(* IEC 61131-3 sources: volt/packages/volt-lsp-iec/test-corpus/pro2193/Device/Plc Logic/Application/99 Library/Function Blocks/JSON builders, 6 files *)

(* ---- BoxFillingJsonFB.pou ---- *)
FUNCTION_BLOCK BoxFillingJsonFB
EXTENDS ToJsonBaseFB
VAR_IN_OUT
	stacks					: ARRAY[1..GVL_Constants_BFU.MaxNumberOfStacksInBox] OF Fanuc_StackPosition;
	boxSettings				: Fanuc_BoxSettings;
	teachPosition			: Fanuc_PositionXYZWPR_Type;
	JSON					: STRING(14000);
END_VAR

%LANGUAGE ST
SUPER^();

IF busy THEN
	IF CreateFinalJson() THEN
		busy		:= FALSE;
		done		:= TRUE;
	END_IF
END_IF

END_FUNCTION_BLOCK

METHOD PRIVATE CreateBoxSettingsJson
VAR_INPUT
	pJson				: POINTER TO STRING(1);
	jsonSize			: UDINT;
END_VAR
VAR_INST
	asProperties		: ARRAY[0..10, 0..1] OF STRING(10);
END_VAR

%LANGUAGE ST
// Fill data
asProperties[0, 0]			:= 'bx';	asProperties[0, 1]			:= TO_STRING(boxSettings.BoxSize.rPosX);
asProperties[1, 0]			:= 'by';	asProperties[1, 1]			:= TO_STRING(boxSettings.BoxSize.rPosY);
asProperties[2, 0]			:= 'bz';	asProperties[2, 1]			:= TO_STRING(boxSettings.BoxSize.rPosZ);
asProperties[3, 0]			:= 'sx';	asProperties[3, 1]			:= TO_STRING(boxSettings.StackSize.rPosX);
asProperties[4, 0]			:= 'sy';	asProperties[4, 1]			:= TO_STRING(boxSettings.StackSize.rPosY);
asProperties[5, 0]			:= 'sz';	asProperties[5, 1]			:= TO_STRING(boxSettings.StackSize.rPosZ);
asProperties[6, 0]			:= 'or';	asProperties[6, 1]			:= TO_STRING(boxSettings.StackOrientation);
asProperties[7, 0]			:= 'sh';	asProperties[7, 1]			:= TO_STRING(boxSettings.StackShape);
asProperties[8, 0]			:= 'tx';	asProperties[8, 1]			:= TO_STRING(teachPosition.rPosX);
asProperties[9, 0]			:= 'ty';	asProperties[9, 1]			:= TO_STRING(teachPosition.rPosY);
asProperties[10, 0]			:= 'tz';	asProperties[10, 1]			:= TO_STRING(teachPosition.rPosZ);

CreateJson(
	psProperties				:= ADR(asProperties),
	udiPropertiesArraySize		:= SIZEOF(asProperties),
	udiPropertiesStringLength	:= SIZEOF(asProperties[0,0]),
	psJSON						:= pJson,
	udiJSONStringLength			:= jsonSize);

END_METHOD

METHOD PRIVATE CreateFinalJson : BOOL
VAR_INST
	asProperties		: ARRAY[0..GVL_Constants_BFU.MaxNumberOfStacksInBox, 0..1] OF STRING(280);
	localJSON			: STRING(14000);
END_VAR

%LANGUAGE ST
sw.Reset();

CASE chunk OF
	0:
		// Create box settings json
		sw.Start();
		asProperties[chunk, 0]	:= 'box';
		CreateBoxSettingsJson(ADR(asProperties[chunk, 1]), SIZEOF(asProperties[chunk, 1]));
		Increment.AnyInt(chunk);
		sw.End();

	1..GVL_Constants_BFU.MaxNumberOfStacksInBox:
		sw.Start();
		asProperties[chunk, 0]	:= CONCAT('S', TO_STRING(chunk));
		CreateStackJson(chunk, ADR(asProperties[chunk, 1]), SIZEOF(asProperties[chunk, 1]));
		Increment.AnyInt(chunk);
		sw.End();

	31:
		Increment.AnyInt(chunk);
	32:
		Increment.AnyInt(chunk);
	33:
		sw.Start();
		CreateJson(
			psProperties				:= ADR(asProperties),
			udiPropertiesArraySize		:= SIZEOF(asProperties),
			udiPropertiesStringLength	:= SIZEOF(asProperties[0,0]),
			psJSON						:= ADR(localJSON),
			udiJSONStringLength			:= SIZEOF(localJSON));
		sw.End();
		Increment.AnyInt(chunk);
	34:
		sw.Start();
		JSON := localJSON;
		sw.End();
		CreateFinalJson					:= TRUE;
END_CASE

END_METHOD

METHOD PRIVATE CreateStackJson
VAR_INPUT
	stack				: UINT;
	pJson				: POINTER TO STRING(1);
	jsonSize			: UDINT;
END_VAR
VAR_INST
	asProperties		: ARRAY[0..13, 0..1] OF STRING(10);
END_VAR

%LANGUAGE ST
// Fill data
asProperties[0, 0]			:= 's';		asProperties[0, 1]			:= TO_STRING(stacks[stack].StackNumber);
asProperties[1, 0]			:= 'x';		asProperties[1, 1]			:= TO_STRING(stacks[stack].PlacePosition.rPosX);
asProperties[2, 0]			:= 'y';		asProperties[2, 1]			:= TO_STRING(stacks[stack].PlacePosition.rPosY);
asProperties[3, 0]			:= 'z';		asProperties[3, 1]			:= TO_STRING(stacks[stack].PlacePosition.rPosZ);
asProperties[4, 0]			:= 'w';		asProperties[4, 1]			:= TO_STRING(stacks[stack].PlacePosition.rPosW);
asProperties[5, 0]			:= 'p';		asProperties[5, 1]			:= TO_STRING(stacks[stack].PlacePosition.rPosP);
asProperties[6, 0]			:= 'r';		asProperties[6, 1]			:= TO_STRING(stacks[stack].PlacePosition.rPosR);
asProperties[7, 0]			:= 'ox';	asProperties[7, 1]			:= TO_STRING(stacks[stack].Offset.rPosX);
asProperties[8, 0]			:= 'oy';	asProperties[8, 1]			:= TO_STRING(stacks[stack].Offset.rPosY);
asProperties[9, 0]			:= 'oz';	asProperties[9, 1]			:= TO_STRING(stacks[stack].Offset.rPosZ);
asProperties[10, 0]			:= 'tx';	asProperties[10, 1]			:= TO_STRING(stacks[stack].ToolOffset.rPosX);
asProperties[11, 0]			:= 'ty';	asProperties[11, 1]			:= TO_STRING(stacks[stack].ToolOffset.rPosY);
asProperties[12, 0]			:= 'tz';	asProperties[12, 1]			:= TO_STRING(stacks[stack].ToolOffset.rPosZ);
asProperties[13, 0]			:= 'c';		asProperties[13, 1]			:= TO_STRING(stacks[stack].Config);

CreateJson(
	psProperties				:= ADR(asProperties),
	udiPropertiesArraySize		:= SIZEOF(asProperties),
	udiPropertiesStringLength	:= SIZEOF(asProperties[0,0]),
	psJSON						:= pJson,
	udiJSONStringLength			:= jsonSize);

END_METHOD

(* ---- CassetteToJsonFB.pou ---- *)
FUNCTION_BLOCK CassetteToJsonFB
EXTENDS ToJsonBaseFB
VAR_INPUT
	CurrentDrawer			: enumDrawer;
END_VAR
VAR_IN_OUT
	CassetteDefinition		: ARRAY[1..GVL_Constants_Magazine.MaxCassettes] OF CassetteDefinition;
	TargetCassettePosition	: ARRAY[enumDrawer.Upper..enumDrawer.Lower, 1..GVL_Constants_Magazine.MaxCassettes] OF CassettePosition;
	DataCassettePosition	: ARRAY[enumDrawer.Upper..enumDrawer.Lower, 1..GVL_Constants_Magazine.MaxCassettes] OF CassettePosition;
	ActualCassettePosition	: ARRAY[enumDrawer.Upper..enumDrawer.Lower, 1..GVL_Constants_Magazine.MaxCassettes] OF CassettePosition;
	JSON					: STRING(25000);
END_VAR

%LANGUAGE ST
SUPER^();

IF busy THEN
	sw.Start();
	IF CreateFinalJson() THEN
		busy		:= FALSE;
		done		:= TRUE;
	END_IF
	sw.End();
END_IF

END_FUNCTION_BLOCK

METHOD PRIVATE CreateCassetteJson
VAR_INPUT
	cassette			: UINT;
	pJson				: POINTER TO STRING(1);
	jsonSize			: UDINT;
END_VAR
VAR_INST
	asProperties		: ARRAY[0..8, 0..1] OF STRING(50);
END_VAR

%LANGUAGE ST
// Fill data
asProperties[0, 0]		:= 'Id';	asProperties[0, 1]		:= TO_STRING(CassetteDefinition[cassette].CassetteId);
asProperties[1, 0]		:= 'Cid';	asProperties[1, 1]		:= TO_STRING(CassetteDefinition[cassette].CavityId);
asProperties[2, 0]		:= 'Lid';	asProperties[2, 1]		:= TO_STRING(CassetteDefinition[cassette].LabelId);
asProperties[3, 0]		:= 'Ltp';	asProperties[3, 1]		:= TO_STRING(CassetteDefinition[cassette].LabelType);
asProperties[4, 0]		:= 'Lor';	asProperties[4, 1]		:= TO_STRING(CassetteDefinition[cassette].LabelOrientation);
asProperties[5, 0]		:= 'Cor';	asProperties[5, 1]		:= TO_STRING(CassetteDefinition[cassette].CassetteOrientation);
asProperties[6, 0]		:= 'Act';	CreatePositionJson(position := ActualCassettePosition[	CurrentDrawer, cassette], ADR(asProperties[6, 1]), SIZEOF(asProperties[6, 1]));
asProperties[7, 0]		:= 'Tgt';	CreatePositionJson(position := TargetCassettePosition[	CurrentDrawer, cassette], ADR(asProperties[7, 1]), SIZEOF(asProperties[7, 1]));
asProperties[8, 0]		:= 'Dat';	CreatePositionJson(position := DataCassettePosition[	CurrentDrawer, cassette], ADR(asProperties[8, 1]), SIZEOF(asProperties[8, 1]));

CreateJson(
	psProperties				:= ADR(asProperties),
	udiPropertiesArraySize		:= SIZEOF(asProperties),
	udiPropertiesStringLength	:= SIZEOF(asProperties[0,0]),
	psJSON						:= pJson,
	udiJSONStringLength			:= jsonSize);

END_METHOD

METHOD PRIVATE CreateFinalJson : BOOL
VAR_INST
	asProperties		: ARRAY[1..GVL_Constants_Magazine.MaxCassettes, 0..1] OF STRING(300);
END_VAR

%LANGUAGE ST
CASE chunk OF
	0:
		Increment.AnyInt(chunk);

	1..GVL_Constants_Magazine.MaxCassettes:
		asProperties[chunk, 0]		:= CONCAT('C', TO_STRING(chunk));
		CreateCassetteJson(chunk, ADR(asProperties[chunk, 1]), SIZEOF(asProperties[chunk, 1]));
		Increment.AnyInt(chunk);

	ELSE
		CreateJson(
			psProperties				:= ADR(asProperties),
			udiPropertiesArraySize		:= SIZEOF(asProperties),
			udiPropertiesStringLength	:= SIZEOF(asProperties[1,0]),
			psJSON						:= ADR(JSON),
			udiJSONStringLength			:= SIZEOF(JSON));

		CreateFinalJson					:= TRUE;
END_CASE

END_METHOD

METHOD PRIVATE CreatePositionJson
VAR_INPUT
	position			: REFERENCE TO CassettePosition;
	pJson				: POINTER TO STRING(1);
	jsonSize			: UDINT;
END_VAR
VAR_INST
	asProperties		: ARRAY[0..2, 0..1] OF STRING(5);
END_VAR

%LANGUAGE ST
//Fill data
asProperties[0,0]		:= 'X1';	asProperties[0,1]		:= TO_STRING(position.X1);
asProperties[1,0]		:= 'X2';	asProperties[1,1]		:= TO_STRING(position.X2);
asProperties[2,0]		:= 'Y';		asProperties[2,1]		:= TO_STRING(position.Y);

CreateJson(
	psProperties				:= ADR(asProperties),
	udiPropertiesArraySize		:= SIZEOF(asProperties),
	udiPropertiesStringLength	:= SIZEOF(asProperties[0,0]),
	psJSON						:= pJson,
	udiJSONStringLength			:= jsonSize);

END_METHOD

(* ---- CavityAliasesToJsonFB.pou ---- *)
FUNCTION_BLOCK CavityAliasesToJsonFB
EXTENDS ToJsonBaseFB
VAR_IN_OUT
	aliases					: ARRAY[GVL_Constants.CavityStartIndex..GVL_Constants.CavityEndIndex] OF STRING(20);
	JSON					: STRING(2000);
END_VAR

%LANGUAGE ST
SUPER^();

IF busy THEN
	sw.Start();
	IF CreateCavityAliasJson() THEN
		busy		:= FALSE;
		done		:= TRUE;
	END_IF
	sw.End();
END_IF

END_FUNCTION_BLOCK

METHOD PRIVATE CreateCavityAliasJson  : BOOL
VAR_INST
	asProperties		: ARRAY[GVL_Constants.CavityStartIndex..GVL_Constants.CavityEndIndex, 0..1] OF STRING(20);
END_VAR

%LANGUAGE ST
// Fill data
FOR chunk := GVL_Constants.CavityStartIndex TO GVL_Constants.CavityEndIndex DO
	asProperties[chunk, 0]			:= TO_STRING(chunk);
	asProperties[chunk, 1]			:= aliases[chunk];
END_FOR

CreateJson(
	psProperties				:= ADR(asProperties),
	udiPropertiesArraySize		:= SIZEOF(asProperties),
	udiPropertiesStringLength	:= SIZEOF(asProperties[GVL_Constants.CavityStartIndex, 0]),
	psJSON						:= ADR(JSON),
	udiJSONStringLength			:= SIZEOF(JSON));

CreateCavityAliasJson			:= TRUE;

END_METHOD

(* ---- RejectReasonAliasesToJsonFB.pou ---- *)
FUNCTION_BLOCK RejectReasonAliasesToJsonFB
EXTENDS ToJsonBaseFB
VAR_IN_OUT
	aliases					: ARRAY[1..GVL_Constants.MaxRejectReasonsTotal] OF STRING(40);
	JSON					: STRING(2000);
END_VAR

%LANGUAGE ST
SUPER^();

IF busy THEN
	sw.Start();
	IF CreateRejectReasonAliasJson() THEN
		busy		:= FALSE;
		done		:= TRUE;
	END_IF
	sw.End();
END_IF

END_FUNCTION_BLOCK

METHOD PRIVATE CreateRejectReasonAliasJson : BOOL
VAR_INST
	asProperties		: ARRAY[1..GVL_Constants.MaxRejectReasonsTotal, 0..1] OF STRING(20);
END_VAR

%LANGUAGE ST
// Fill data
FOR chunk := 1 TO GVL_Constants.MaxRejectReasonsTotal DO
	asProperties[chunk, 0]			:= TO_STRING(chunk);
	asProperties[chunk, 1]			:= aliases[chunk];
END_FOR

CreateJson(
	psProperties				:= ADR(asProperties),
	udiPropertiesArraySize		:= SIZEOF(asProperties),
	udiPropertiesStringLength	:= SIZEOF(asProperties[1, 0]),
	psJSON						:= ADR(JSON),
	udiJSONStringLength			:= SIZEOF(JSON));

CreateRejectReasonAliasJson		:= TRUE;

END_METHOD

(* ---- StatsToJsonFB.pou ---- *)
FUNCTION_BLOCK StatsToJsonFB
EXTENDS ToJsonBaseFB
VAR_IN_OUT
	stats					: ProductionStatsType;
	JSON					: STRING(25000);
END_VAR

%LANGUAGE ST
SUPER^();

IF busy THEN
	sw.Start();
	IF CreateFinalJson() THEN
		busy		:= FALSE;
		done		:= TRUE;
	END_IF
	sw.End();
END_IF

END_FUNCTION_BLOCK

METHOD PRIVATE CreateFinalJson : BOOL
VAR_INST
	asProperties		: ARRAY[1..GVL_Constants.MaxProductsInMould + 2, 0..1] OF STRING(1000);
END_VAR

%LANGUAGE ST
CASE chunk OF
	0:
		Increment.AnyInt(chunk);

	1..GVL_Constants.MaxProductsInMould:
		asProperties[chunk, 0]	:= CONCAT('C', TO_STRING(chunk));
		CreateProductionStatsCavityJson(stat := stats.Cavity[chunk], pJson := ADR(asProperties[chunk, 1]), jsonSize := SIZEOF(asProperties[chunk, 1]));
		Increment.AnyInt(chunk);

	ELSE
		IF chunk = GVL_Constants.MaxProductsInMould + 1 THEN
			asProperties[chunk, 0]	:= 'T';
			CreateProductionStatsCavityJson(stat := stats.Total, pJson := ADR(asProperties[chunk, 1]), jsonSize := SIZEOF(asProperties[chunk, 1]));
			Increment.AnyInt(chunk);
		ELSIF chunk = GVL_Constants.MaxProductsInMould + 2 THEN
			asProperties[chunk, 0]	:= 'S';
			CreateTimerJson(pJson := ADR(asProperties[chunk, 1]), jsonSize := SIZEOF(asProperties[chunk, 1]));
			Increment.AnyInt(chunk);
		ELSE
			CreateJson(
				psProperties				:= ADR(asProperties),
				udiPropertiesArraySize		:= SIZEOF(asProperties),
				udiPropertiesStringLength	:= SIZEOF(asProperties[1,0]),
				psJSON						:= ADR(JSON),
				udiJSONStringLength			:= SIZEOF(JSON));

			CreateFinalJson					:= TRUE;
		END_IF
END_CASE

END_METHOD

METHOD PRIVATE CreateProductionStatsCavityJson
VAR_INPUT
	pJson : POINTER TO STRING(1);
	jsonSize : UDINT;
END_VAR
VAR_IN_OUT
	stat				: ProductionStatsCavityType;
END_VAR
VAR_INST
	asProperties		: ARRAY[0..GVL_Constants.MaxRejectReasonsTotal + 3, 0..1] OF STRING(25);
	i					: UINT;
END_VAR

%LANGUAGE ST
// Fill data
asProperties[0, 0]	:= 'P';		asProperties[0, 1] := TO_STRING(stat.Produced);
asProperties[1, 0]	:= 'S';		asProperties[1, 1] := TO_STRING(stat.Stacked);
asProperties[2, 0]	:= 'R';		asProperties[2, 1] := TO_STRING(stat.Rejected);
asProperties[3, 0]	:= 'U';		asProperties[3, 1] := TO_STRING(stat.UncountedReject);

FOR i := 4 TO GVL_Constants.MaxRejectReasonsTotal + 3 DO
	asProperties[i, 0]	:= CONCAT('R', TO_STRING(i - 3));
	asProperties[i, 1]	:= TO_STRING(stat.RejectReason[i - 3]);
END_FOR

CreateJson(
	psProperties				:= ADR(asProperties),
	udiPropertiesArraySize		:= SIZEOF(asProperties),
	udiPropertiesStringLength	:= SIZEOF(asProperties[0,0]),
	psJSON						:= pJson,
	udiJSONStringLength			:= jsonSize);

END_METHOD

METHOD PRIVATE CreateTimerJson
VAR_INPUT
	pJson				: POINTER TO STRING(1);
	jsonSize			: UDINT;
END_VAR
VAR_INST
	asProperties		: ARRAY[0..5, 0..1] OF STRING(25);
END_VAR

%LANGUAGE ST
// Fill data
asProperties[0, 0]		:= 'N';		asProperties[0, 1]		:= TO_STRING(stats.StatId);
asProperties[1, 0]		:= 'S';		asProperties[1, 1]		:= TO_STRING(stats.TimeStopped);
asProperties[2, 0]		:= 'R';		asProperties[2, 1]		:= TO_STRING(stats.TimeResetting);
asProperties[3, 0]		:= 'I';		asProperties[3, 1]		:= TO_STRING(stats.TimeIdle);
asProperties[4, 0]		:= 'A';		asProperties[4, 1]		:= TO_STRING(stats.TimeAutomatic);
asProperties[5, 0]		:= 'C';		asProperties[5, 1]		:= TO_STRING(stats.AutomaticCycleStarts);

CreateJson(
	psProperties				:= ADR(asProperties),
	udiPropertiesArraySize		:= SIZEOF(asProperties),
	udiPropertiesStringLength	:= SIZEOF(asProperties[0,0]),
	psJSON						:= pJson,
	udiJSONStringLength			:= jsonSize);

END_METHOD

(* ---- ToJsonBaseFB.pou ---- *)
FUNCTION_BLOCK ABSTRACT ToJsonBaseFB
VAR_INPUT
	execute					: BOOL;
END_VAR
VAR_OUTPUT
	busy					: BOOL;
	done					: BOOL;
END_VAR
VAR
	chunk					: UINT;
	sw						: StopwatchFB;
END_VAR

%LANGUAGE ST
IF execute THEN
	IF NOT busy THEN
		chunk		:= 0;
	END_IF
	busy			S= NOT done;
ELSE
	done			:= FALSE;
END_IF

END_FUNCTION_BLOCK

METHOD PROTECTED CreateJson
VAR_INPUT
	psProperties				: POINTER TO STRING(1);		// Double array: key/value [0..*,0..1]
	udiPropertiesArraySize		: UDINT;					// Total size of array
	udiPropertiesStringLength	: UDINT;					// Length of string (key/value)
	psJSON						: POINTER TO STRING(1);		// Output for content
	udiJSONStringLength			: UDINT;					// Length of string
END_VAR
VAR_INST
	JSON_builder			: L_ITCA_JSON_Builder_Variable;
END_VAR

// L_ITCA_JSON_Builder_Variable FB always finishes the same PLC cycle.
// It could actually be a Function instead
// JSON libs received from Lenze and stored here: N:\Software\Automation\Lenze\Libraries\Lenze JSON lib

%LANGUAGE ST
// Create content
JSON_builder(
	xExecute					:= TRUE,
	psProperties				:= psProperties,
	udiPropertiesArraySize		:= udiPropertiesArraySize,
	udiPropertiesStringLength	:= udiPropertiesStringLength,
	psJSON						:= psJSON,
	udiJSONStringLength			:= udiJSONStringLength);

JSON_builder(
	xExecute					:= FALSE);

END_METHOD

// Enables the FB to recreate the JSON while execute input remains high
METHOD PUBLIC Reset

%LANGUAGE ST
busy	:= FALSE;
done	:= FALSE;

END_METHOD
